Staubli VAL3: ros2_server.pjx

--- ros2_server.pjx ---
Parameters version=s8.20.2Cs9_BS4270 stackSize=5000 millimeterUnit=true
Program file=Comm/computeSequenceDelay.pgx
Program file=Comm/getNextSequenceNumber.pgx
Program file=Comm/readData.pgx
Program file=Comm/readDataOnce.pgx
Program file=Comm/resetControlSocket.pgx
Program file=Comm/sendData.pgx
Program file=Control/stopJointPositionControl.pgx
Program file=Control/stopJointVelocityControl.pgx
Program file=Control/updateJointPositionControl.pgx
Program file=Control/updateJointVelocityControl.pgx
Program file=controlTask.pgx
Program file=Serialization/decodeHeader.pgx
Program file=Serialization/decodeRobotCommandMsg.pgx
Program file=Serialization/encodeHeader.pgx
Program file=Serialization/encodeRobotStateMsg.pgx
Program file=Serialization/initHeader.pgx
Program file=Serialization/initRobotCommandMsg.pgx
Program file=Serialization/initRobotStateMsg.pgx
Program file=Utils/logThrottleMsg.pgx
Program file=start.pgx
Program file=stop.pgx
Program file=updateState.pgx
Data file=ros2_server.dtx
Type name=ThrottleLogMsg path=Disk://ros2_server/Types/ThrottleLogMsg/ThrottleLogMsg.pjx
Type name=MessageHeader path=Disk://ros2_server/Types/MessageHeader/MessageHeader.pjx
Type name=RobotState path=Disk://ros2_server/Types/RobotState/RobotState.pjx
Type name=RobotStateMsg path=Disk://ros2_server/Types/RobotStateMsg/RobotStateMsg.pjx
Type name=RobotCommand path=Disk://ros2_server/Types/RobotCommand/RobotCommand.pjx
Type name=RobotCommandMsg path=Disk://ros2_server/Types/RobotCommandMsg/RobotCommandMsg.pjx

--- ros2_server.dtx ---
public sio siSocketControl = {link=UdpSocket\fuzzyudp}
public bool bIsOverrun = true
mdesc mMdesc = {blend=off}
public num nErrorCode
public num nInError
public num nOverruns

--- start.pgx ---
program start()
  local string l_sVal3
  local string l_sMajor
  local num l_nCtrlPeriod
  local num l_nBoxcarDelay
begin
  logMsg("ros2_server::start : starting application")

  // Get VAL3 version
  l_sVal3=getVersion("System")
  l_sMajor=mid(l_sVal3,1,1)

  // Check boxcar filter configuration
  //$setBoxcarFreq(60.0)
  l_nBoxcarDelay = $getBoxcarDelay()
  logMsg("ros2_server::start : boxcar delay is " + toString("0.1",l_nBoxcarDelay), 1)

  // Speed must be at 100%
  if getMonitorSpeed()<100
    logMsg("ros2_server::start : Warning, monitor speed is below 100% and control algorithms might not work correctly...", 2)
    // popUpMsg("The monitor speed must be at 100%, waiting...")
    // wait(getMonitorSpeed() == 100)
  endIf

  // Reset socket buffers
  clearBuffer(siSocketControl)

  // Setup supervision/diagnostics task
  // TODO

  // Setup control task
  l_nCtrlPeriod = 0.004
  mMdesc.blend = off

  stopMove()
  resetMotion()
  autoConnectMove(true)

  // Start control task
  bIsOverrun = false
  taskCreateSync "controlTask", l_nCtrlPeriod, bIsOverrun, controlTask()
end

--- controlTask.pgx ---
program controlTask()
  local bool l_bError
  local bool l_bErrorTmp
  local bool l_bRxError
  local bool l_bPreviousRxError
  local bool l_bTxError
  local num l_nSequenceNumber
  local num l_nSequenceDelay
  local RobotStateMsg robot_state_msg
  local RobotCommandMsg robot_command_msg
  local num l_nCmdMode
  local num l_nPreviousCmdMode
  local bool l_bNewCmdMessage
  local bool l_bStopControlTask
  local bool l_bControlActive
  local ThrottleLogMsg throttle_sequence_delay_msg
begin
  popUpMsg("ros2_server::controlTask : Initializing control task")
  l_bStopControlTask = false
  // Reset errors
  l_bError = false
  l_bErrorTmp = false
  l_bControlActive = false
  nOverruns = 0
  l_nSequenceNumber = 0
  l_nSequenceDelay = 1000

  // Reset command mode (STOP)
  // Implemented modes :
  // 0 : Invalid / Error
  // 1 : STOP / Idle
  // 2 : Joint position control
  // 3 : Joint velocity control
  l_nCmdMode = 1
  l_nPreviousCmdMode = 1

  // Initialize robot state message
  call initRobotStateMsg(robot_state_msg, l_bErrorTmp)
  if(l_bErrorTmp)
    l_bError = true
    logMsg("ros2_server::controlTask : Error, failed to init robot state msg", 3)
    return
  endIf

  // Initialize robot command message
  call initRobotCommandMsg(robot_command_msg, l_bErrorTmp)
  if(l_bErrorTmp)
    l_bError = true
    logMsg("ros2_server::controlTask : Error, failed to init robot command msg", 3)
    return
  endIf

  // Initialize control socket
  call resetControlSocket(siSocketControl, l_bErrorTmp)
  if(l_bErrorTmp)
    l_bError = true
    logMsg("ros2_server::controlTask : Error, failed to reset socket", 3)
    return
  endIf

  // Initialize throttle log msg for sequence delay warnings
  throttle_sequence_delay_msg.sMsg = "ros2_server::controlTask : communication latency detected! "
  throttle_sequence_delay_msg.nThrottleInterval = 10.0
  throttle_sequence_delay_msg.nSeverity = 2

  // Main control loop
  popUpMsg("ros2_server::controlTask : Starting control task")
  while !l_bStopControlTask
    // Check for task overrun
    if bIsOverrun
      logMsg("ros2_server::controlTask : Task overrun detected", 2)
      bIsOverrun = false
      nOverruns = nOverruns + 1
    endIf
    // -------------------------------
    // Update and publish robot state
    // -------------------------------

    // Update robot state
    call updateState(robot_state_msg.robotState)

    // Update sequence number
    call getNextSequenceNumber(l_nSequenceNumber)
    robot_state_msg.header.nMsgSequenceNumber = l_nSequenceNumber
    robot_state_msg.robotState.nSequenceDelay = l_nSequenceDelay

    // Check for errors that would require a hard stop now
    // Robot is moving when it shouldn't
    // TODO
    // Warning emergency stop pressed
    // TODO
    // Runtime errors
    // TODO

    // Update control state
    robot_state_msg.robotState.bInError = l_bError
    robot_state_msg.robotState.nControlMode = l_nCmdMode
    // Publish robot state
    l_bTxError = false
    call encodeRobotStateMsg(robot_state_msg, l_bTxError)
    if(!l_bTxError)
      call sendData(siSocketControl, robot_state_msg.nSerializedData, l_bTxError)
    endIf
    if(l_bTxError)
      logMsg("ros2_server::controlTask : Failed to encode/send robot state", 2)
      l_bError = true
    endIf

    // -------------------------------
    // Receive and process command
    // -------------------------------
    // (Try to) read the last command msg
    call readData(siSocketControl, robot_command_msg.nSerializedData, l_bNewCmdMessage, l_bRxError)

    if(l_bRxError)
      logMsg("ros2_server::controlTask : error during command msg read", 2)
      l_bError = true
    else
      // New data received?
      if(l_bNewCmdMessage)
        call decodeRobotCommandMsg(robot_command_msg, l_bErrorTmp)
        if(l_bErrorTmp)
          logMsg("ros2_server::controlTask : Error, failed to decode command msg", 3)
          // Flag fatal error and go to STOP mode
          l_bError = true
          l_nCmdMode = 1
        endIf
      elseIf(robot_command_msg.robotCommand.bIsValid)
        // No new message, check staleness of previous message
        // TODO
      endIf
    endIf

    if (l_bNewCmdMessage and !l_bControlActive)
      l_bControlActive = true
      logMsg("ros2_server::controlTask : connection to controller established", 1)
    endIf

    // Check stream (staleness, lost pkg, etc.)
    if (robot_command_msg.robotCommand.bIsValid)
      call computeSequenceDelay(l_nSequenceNumber, robot_command_msg.header.nMsgSequenceNumber, l_nSequenceDelay)
    else
      // No valid command received yet, set arbitrary large delay
      l_nSequenceDelay = 1000
    endIf

    if (l_bControlActive)
      // Log warning if a ping-pong delay is above two control cycles
      if (l_nSequenceDelay > 3)
        call logThrottleMsg(throttle_sequence_delay_msg)
      endIf
      // Error case 1: robot is moving -> fatal error if delay too high (>20ms)
      // TODO: modulate acceptable limit depending on control mode (i.e., smaller for velocity...)
      if (robot_state_msg.robotState.bInMotion and l_nSequenceDelay > 5)
        logMsg("ros2_server::controlTask : Error, command sequence delay too high during robot motion (" + toString("0.1", l_nSequenceDelay) + "), going to STOP mode", 3)
        l_bError = true
        l_nCmdMode = 1
      endIf
      // Error case 2: robot is not moving -> allow up to 100ms delay before error as there is no actual risk
      if (!robot_state_msg.robotState.bInMotion and l_nSequenceDelay > 25)
        logMsg("ros2_server::controlTask : Error, command sequence delay too high (" + toString("0.1", l_nSequenceDelay) + "), going to STOP mode", 3)
        l_bError = true
        l_nCmdMode = 1
      endIf
      // Check for negative delay (should not happen)
      if (l_nSequenceDelay < 0)
        logMsg("ros2_server::controlTask : Error, negative command sequence delay, going to STOP mode", 3)
        l_bError = true
        l_nCmdMode = 1
      endIf
    endIf

    // Check command type validity
    if (robot_command_msg.robotCommand.nMotionCmdType < 0 or robot_command_msg.robotCommand.nMotionCmdType > 4)
      logMsg("ros2_server::controlTask : Error, invalid command mode", 2)
      robot_command_msg.robotCommand.bIsValid = false
      l_bError = true
    endIf
    // TODO: staleness, lost pkg, etc.

    // Extract command mode
    if (l_bError or !robot_command_msg.robotCommand.bIsValid)
      // In case of error, go to ERROR mode
      l_nCmdMode = 0
    else
      l_nCmdMode = robot_command_msg.robotCommand.nMotionCmdType
    endIf

    // Check command transition validity
    if(l_nPreviousCmdMode != l_nCmdMode and l_nCmdMode != 1 and l_nPreviousCmdMode != 1)
      // Transitioning from a command mode to another requires a stop
      l_nCmdMode = 1
      l_bError = true
      logMsg("ros2_server::controlTask : Error, transitioning from command modes requires a stop", 2)
    endIf

    if (l_nPreviousCmdMode == 1 and l_nCmdMode != 1 and robot_state_msg.robotState.bInMotion)
      // Robot is still moving from previous command, cannot start new command yet
      l_nCmdMode = 1
      logMsg("ros2_server::controlTask : Warning, robot still in motion, cannot start new command yet", 2)
      l_bError = true
    endIf

    // -------------------------------
    // Execute motion command
    // -------------------------------
    if(l_nCmdMode <= 1)
      // -------------------------------
      // Execute STOP command (or ERROR)
      // -------------------------------
      if(l_nPreviousCmdMode == 2)
        logMsg("ros2_server::controlTask : Stopping joint position command mode", 1)
        call stopJointPositionControl(l_bErrorTmp)
        if(l_bErrorTmp)
          l_bError = true
          logMsg("ros2_server::controlTask : Error, failed to stop joint position control", 2)
        endIf
      elseIf(l_nPreviousCmdMode == 3)
        logMsg("ros2_server::controlTask : Stopping joint velocity command mode", 1)
        call stopJointVelocityControl(l_bErrorTmp)
        if(l_bErrorTmp)
          l_bError = true
          logMsg("ros2_server::controlTask : Error, failed to stop joint velocity control", 2)
        endIf
      endIf
      // Stop / wait for new command
      stopMove()
      resetMotion()
    elseIf(l_nCmdMode == 2)
      // -------------------------------
      // Execute joint position command
      // -------------------------------
      if(l_nPreviousCmdMode == 1)
        logMsg("ros2_server::controlTask : Starting joint position command mode", 1)
        call updateJointPositionControl(robot_state_msg.robotState, robot_command_msg.robotCommand, l_bErrorTmp, true)
      else
        // Continuing in position control mode
        call updateJointPositionControl(robot_state_msg.robotState, robot_command_msg.robotCommand, l_bErrorTmp, false)
      endIf
      if(l_bErrorTmp)
        l_bError = true
        logMsg("ros2_server::controlTask : Error, failed to update joint position control", 2)
      endIf
    elseIf(l_nCmdMode == 3)
      // -------------------------------
      // Execute joint velocity command
      // -------------------------------
      if(l_nPreviousCmdMode == 1)
        logMsg("ros2_server::controlTask : Starting joint velocity command mode", 1)
        call updateJointVelocityControl(robot_state_msg.robotState, robot_command_msg.robotCommand, l_bErrorTmp, true)
      else
        // Continuing in velocity control mode
        call updateJointVelocityControl(robot_state_msg.robotState, robot_command_msg.robotCommand, l_bErrorTmp, false)
      endIf
      if(l_bErrorTmp)
        l_bError = true
        logMsg("ros2_server::controlTask : Error, failed to update joint velocity control", 2)
      endIf
    else
      // -------------------------------
      // Handle invalid motion command
      // -------------------------------
      logMsg("ros2_server::controlTask : Unknown command mode", 2)
      l_bError = true
    endIf

    // -------------------------------
    // Execute GPIO commands
    // -------------------------------
    // TODO: write digital outputs based on command
    // TODO: write analog outputs based on command

    // -------------------------------
    // Handle errors
    // -------------------------------
    if(l_bError)
      logMsg("ros2_server::controlTask : Error, hard stop and reset", 3)

      // Stop motion
      if (l_nCmdMode == 2)
        logMsg("ros2_server::controlTask : Stopping joint position command mode due to error", 1)
        call stopJointPositionControl(l_bErrorTmp)
        if(l_bErrorTmp)
          logMsg("ros2_server::controlTask : Error, failed to stop joint position control", 2)
        endIf
      endIf

      stopMove()
      resetMotion()
      robot_command_msg.robotCommand.nMotionCmdType = 0
      l_nCmdMode = 0

      // Clear flag and reset communication
      l_bError = false

      l_nSequenceNumber=0
      l_nSequenceDelay = 1000
      l_bTxError = false
      l_bRxError = false
      l_bPreviousRxError = false
      l_bControlActive = false
      robot_command_msg.robotCommand.bIsValid = false
      call resetControlSocket(siSocketControl, l_bErrorTmp)
      if(l_bErrorTmp)
        logMsg("ros2_server::controlTask : Error, failed to reset socket")
        l_bError = true
      endIf

      // TODO: add delay (e.g., 1000ms) before accepting new commands?
    endIf

    // -------------------------------
    // Prepare for next iteration
    // -------------------------------
    l_nPreviousCmdMode = l_nCmdMode
    l_bPreviousRxError = l_bRxError

    // Sleep until next period
    delay(0)
    // -------------------------------
  endWhile

  // Cleanup
  logMsg("ros2_server::controlTask : Stopping Control Loop")
  stopMove()
  resetMotion()
end

--- stop.pgx ---
program stop()
begin
  logMsg("ros2_server::stop : quitting application")
  // Stop motion
  stopMove()
  resetMotion()
  // Clear socket buffers
  clearBuffer(siSocketControl)
end

--- updateState.pgx ---
public program updateState(RobotState& x_state)
  local num l_nJntVelArray[6]
  local num l_nJntTorqueArray[6]
  local num l_nEStopStatus
begin
  // Read the robot state and fill the RobotState structure
  // Sets "x_state.bIsValid" to true if successful, false otherwise
  // Note that some fields should be filled by the caller:
  // - bInError
  // - nSequenceDelay
  // - nControlMode (Stop / Position / Velocity / etc. )
  x_state.bIsValid = false

  // -------------------------
  // Fill status fields
  // -------------------------
  // Power and motion
  x_state.bDrivePowered = isPowered()
  x_state.bBrakeReleased = x_state.bDrivePowered
  x_state.bInMotion = !isSettled()

  // Safety
  // Estop status:
  //  - 0 No safety stop
  //  - 1 Waiting safety Restart
  //  - 2 SS1 - Safety stop condition
  //  - 3 SS2 - Safe operating stop condition
  //  - 4 Waiting restart from WMS
  x_state.nSafetyStatus = esStatus()
  x_state.bEStopped = (x_state.nSafetyStatus != 0)
  x_state.bWaitAck = (x_state.nSafetyStatus == 1)


  // Robot working mode
  //   0: Invalid / Transition from safety
  //   1: Manual
  //   2: Test
  //   3: Automatic - Local
  //   4: Automatic - Remote
  // The returned status depends on the mode...
  // For automatic modes (3 and 4), status is:
  //   0 : Move (programmed movement)
  //   1 : Move (connection movement)
  //   2 : Hold
  x_state.nRobotMode = workingMode(x_state.nRobotStatus)

  // Motion possible
  x_state.bMotionPossible = (x_state.bDrivePowered and (!x_state.bEStopped))
  // x_state.bMotionPossible = (x_state.bDrivePowered and (!x_state.bEStopped) and (x_state.nRobotStatus == 0))

  // -------------------------
  // Fill joint state
  // -------------------------
  x_state.bValidPosition = true
  x_state.bValidVelocity = true
  x_state.bValidTorque = true

  // Get the current joint positions
  x_state.jointPositions = herej()

  // Get the current joint velocities (approximation)
  $getJntSpeedCmd(l_nJntVelArray)
  x_state.jointVelocities.j1 = l_nJntVelArray[0]
  x_state.jointVelocities.j2 = l_nJntVelArray[1]
  x_state.jointVelocities.j3 = l_nJntVelArray[2]
  x_state.jointVelocities.j4 = l_nJntVelArray[3]
  x_state.jointVelocities.j5 = l_nJntVelArray[4]
  x_state.jointVelocities.j6 = l_nJntVelArray[5]

  // Get the estimated joint torques
  // Note: current joint torque (N.m for revolute axis) or force (N for linear axis) computed from the motors currents.
  // The joint force is not a direct estimation of external efforts. It also includes gravity, friction, viscosity,
  // inertia, noise and accuracy of current sensors, relation between motor current and torque.
  // It returns only an order of magnitude for forces.
  // There is NO COMMITMENT ON ACCURACY!
  getJointForce(l_nJntTorqueArray)
  x_state.jointTorques.j1 = l_nJntTorqueArray[0]
  x_state.jointTorques.j2 = l_nJntTorqueArray[1]
  x_state.jointTorques.j3 = l_nJntTorqueArray[2]
  x_state.jointTorques.j4 = l_nJntTorqueArray[3]
  x_state.jointTorques.j5 = l_nJntTorqueArray[4]
  x_state.jointTorques.j6 = l_nJntTorqueArray[5]

  // -------------------------
  // Fill F/T sensor data (opt.)
  // -------------------------
  // Not implemented
  x_state.bValidFtSensor = false
  x_state.nFtSensorValues[0] = 0.0
  x_state.nFtSensorValues[1] = 0.0
  x_state.nFtSensorValues[2] = 0.0
  x_state.nFtSensorValues[3] = 0.0
  x_state.nFtSensorValues[4] = 0.0
  x_state.nFtSensorValues[5] = 0.0

  // -------------------------
  // Fill IOs state
  // -------------------------
  x_state.bValidDigitalInputs = false
  x_state.bValidAnalogInputs = false

  // -------------------------
  x_state.bIsValid = true
end
